Universal Robots PolyScope program: despellatizing.urp

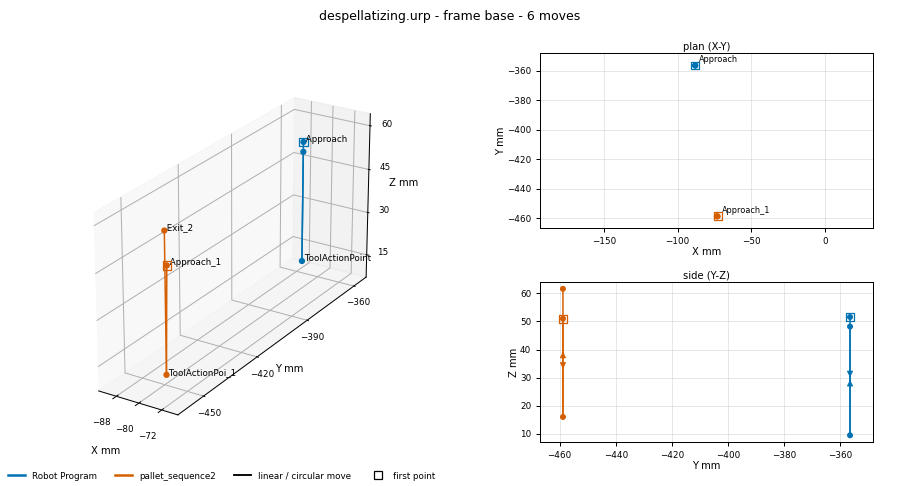
[picture p0: tool path of despellatizing.urp in frame base, 6 of 6 moves have a stored position in this frame; points joined in program order, loops and branches not executed]
Program despellatizing (installation=default ventosa directory=/programs/usbdisk/Ventosa-paleta createdIn=5.12.1.1101497 lastSavedIn=5.12.1.1101497 robotSerialNumber=20225300640)
Calibrated DH parameters: a=[-0.000125, -0.240482, -0.204397, 0.000169, -0.000135, 0]; d=[0.152056, 4.760815, 12.138494, -16.768367, 0.085457, 0.092357]; alpha=[1.570863, 0.008548, 0.003635, 1.571424, -1.571918, 0]; deltaTheta=[0, 0.167622, 0.124346, -0.291972, 0.000034, 0]
BeforeStart
  SafeHome (positionOptionType=SPEED_AND_ACCELERATION speed=1.047198 acceleration=1.396263 nextMotionTime=2)
  cnt_obj := 0
Robot Program (runOnlyOnce=true)
  Loop While (checkContinuously=false) expression=cnt_obj<2
    URCap Palletizing (polyscope-pallet-impl, Universal Robots) dataModel(palletFeature=Base, isPalletizing=false, Variable(key=name, variable(name=Pallet_1)), Variable(key=globalCountingVariable, variable(name=Pallet_1_cnt, initializeExpression=1)), Variable(key=layerNumberVariable, variable(name=Pallet_1_lno, initializeExpression=1)), Variable(key=layerCountingVariable, variable(name=Pallet_1_lct, initializeExpression=1)), Variable(key=handleSeparatorVariable, variable(name=Pallet_1_sep, initializeExpression=False)), Variable(key=totalCountVariable, variable(name=Pallet_1_tct, initializeExpression=1)), Variable(key=referencePoint, variable(featureName=referencePoint)), Variable(key=separatorPoint, variable(featureName=separatorPoint)), Length(key=objectHeight value=0.02 unit=M)); state(isChildrenLocked=true)
      URCap Patterns (polyscope-pallet-impl, Universal Robots) state(isChildrenLocked=true)
        URCap Pattern (polyscope-pallet-impl, Universal Robots) dataModel(UUID=4f81d8ba-079c-47d5-9963-bf25775c8eb8, patternType=LINE, objects=3, Variable(key=nameVariable, variable(name=Line_Pattern_1))); state(isChildrenLocked=true)
          URCap Item (polyscope-pallet-impl, Universal Robots) dataModel(UUID=1e3ca6f4-2eef-47f5-9254-e2ca323da8c7, patternType=LINE, index=0, calibrationDeltaTheta=[-4.022425301349053E-7, 0.1676224840059082, 0.12434612800300923, -0.29197201232783093, 3.427063592260221E-5, -2.1055269264214083E-9], calibrationA=[-1.2536318386722594E-4, -0.24048217598078755, -0.20439712606180582, 1.6856812341359539E-4, -1.3512489031768148E-4, 0.0], calibrationD=[0.1520559623222255, 4.760815016703785, 12.138493934059257, -16.768366633975226, 0.08545691164632878, 0.09235657960129308], calibrationAlpha=[1.570862629498801, 0.008547662301921876, 0.0036353825850200293, 1.5714242532258311, -1.5719182813352055, 0.0], calibrationJointChecksum=[-1442419114, -1443167645, -1459096000, -1465254611, -1461595521, -1465327861], calibrationStatus=2, calibrationValidChecksum=true, baseToFeature=[0.0, 0.0, 0.0, 0.0, 0.0, 0.0], TCPOffset=[-3.1361648691191624E-6, -7.165658321095503E-6, 0.14500622770334937, -3.159826595633942E-6, 1.3472828827308191E-6, -1.5977345697242604E-5], Variable(key=variable, variable(name=StartItem_1)), JointPositions(key=jointpositions, JointPosition(key=[1], Angle(key=pos value=0.956268 unit=RAD)), JointPosition(key=[2], Angle(key=pos value=-1.20615 unit=RAD)), JointPosition(key=[3], Angle(key=pos value=1.878719 unit=RAD)), JointPosition(key=[4], Angle(key=pos value=-2.25283 unit=RAD)), JointPosition(key=[5], Angle(key=pos value=-1.545112 unit=RAD)), JointPosition(key=[6], Angle(key=pos value=-0.610524 unit=RAD))))
          URCap Item (polyscope-pallet-impl, Universal Robots) dataModel(UUID=6f3f843f-6f96-4607-877d-a96ceec1e152, patternType=LINE, index=1, calibrationDeltaTheta=[-4.022425301349053E-7, 0.1676224840059082, 0.12434612800300923, -0.29197201232783093, 3.427063592260221E-5, -2.1055269264214083E-9], calibrationA=[-1.2536318386722594E-4, -0.24048217598078755, -0.20439712606180582, 1.6856812341359539E-4, -1.3512489031768148E-4, 0.0], calibrationD=[0.1520559623222255, 4.760815016703785, 12.138493934059257, -16.768366633975226, 0.08545691164632878, 0.09235657960129308], calibrationAlpha=[1.570862629498801, 0.008547662301921876, 0.0036353825850200293, 1.5714242532258311, -1.5719182813352055, 0.0], calibrationJointChecksum=[-1442419114, -1443167645, -1459096000, -1465254611, -1461595521, -1465327861], calibrationStatus=2, calibrationValidChecksum=true, baseToFeature=[0.0, 0.0, 0.0, 0.0, 0.0, 0.0], TCPOffset=[-8.933406672184674E-6, 6.908638976621528E-6, 0.14500541786871218, -1.4995112137550501E-5, -1.239510916399233E-6, -2.697305733370411E-5], Variable(key=variable, variable(name=EndItem_1)), JointPositions(key=jointpositions, JointPosition(key=[1], Angle(key=pos value=1.450295 unit=RAD)), JointPosition(key=[2], Angle(key=pos value=-1.189136 unit=RAD)), JointPosition(key=[3], Angle(key=pos value=1.845346 unit=RAD)), JointPosition(key=[4], Angle(key=pos value=-2.243967 unit=RAD)), JointPosition(key=[5], Angle(key=pos value=-1.548882 unit=RAD)), JointPosition(key=[6], Angle(key=pos value=-0.116345 unit=RAD))))
      URCap Layers (polyscope-pallet-impl, Universal Robots) dataModel(separators=[false], selectedPatterns=[4f81d8ba-079c-47d5-9963-bf25775c8eb8])
      URCap At Each Item (polyscope-pallet-impl, Universal Robots) dataModel(selectedPattern=4f81d8ba-079c-47d5-9963-bf25775c8eb8, selectedPosition=1e3ca6f4-2eef-47f5-9254-e2ca323da8c7, Approach_calibrationDeltaTheta=[-4.022425301349053E-7, 0.1676224840059082, 0.12434612800300923, -0.29197201232783093, 3.427063592260221E-5, -2.1055269264214083E-9], Approach_calibrationA=[-1.2536318386722594E-4, -0.24048217598078755, -0.20439712606180582, 1.6856812341359539E-4, -1.3512489031768148E-4, 0.0], Approach_calibrationD=[0.1520559623222255, 4.760815016703785, 12.138493934059257, -16.768366633975226, 0.08545691164632878, 0.09235657960129308], Approach_calibrationAlpha=[1.570862629498801, 0.008547662301921876, 0.0036353825850200293, 1.5714242532258311, -1.5719182813352055, 0.0], Approach_calibrationJointChecksum=[-1442419114, -1443167645, -1459096000, -1465254611, -1461595521, -1465327861], Approach_calibrationStatus=2, Approach_calibrationValidChecksum=true, Approach_baseToFeature=[0.0, 0.0, 0.0, 0.0, 0.0, 0.0], Approach_TCPOffset=[-9.367263874154874E-6, -3.571446355488117E-6, 0.1449987796699207, 2.480276054203756E-5, -1.6285190499819042E-5, -2.849487153099717E-6], Exit_calibrationDeltaTheta=[-4.022425301349053E-7, 0.1676224840059082, 0.12434612800300923, -0.29197201232783093, 3.427063592260221E-5, -2.1055269264214083E-9], Exit_calibrationA=[-1.2536318386722594E-4, -0.24048217598078755, -0.20439712606180582, 1.6856812341359539E-4, -1.3512489031768148E-4, 0.0], Exit_calibrationD=[0.1520559623222255, 4.760815016703785, 12.138493934059257, -16.768366633975226, 0.08545691164632878, 0.09235657960129308], Exit_calibrationAlpha=[1.570862629498801, 0.008547662301921876, 0.0036353825850200293, 1.5714242532258311, -1.5719182813352055, 0.0], Exit_calibrationJointChecksum=[-1442419114, -1443167645, -1459096000, -1465254611, -1461595521, -1465327861], Exit_calibrationStatus=2, Exit_calibrationValidChecksum=true, Exit_baseToFeature=[0.0, 0.0, 0.0, 0.0, 0.0, 0.0], Exit_TCPOffset=[-1.637346477856294E-5, 4.478754114078942E-6, 0.14501055095189264, -4.558640450482124E-5, -2.3885119760789442E-6, -5.824444254552941E-5], currentWizardState=LANDING, Pose(key=refBaseToFeature, Position(key=posePosition, Length(key=X value=0 unit=M), Length(key=Y value=0 unit=M), Length(key=Z value=0 unit=M)), Rotation(key=poseRotation, Angle(key=RX value=0 unit=RAD), Angle(key=RY value=0 unit=RAD), Angle(key=RZ value=0 unit=RAD))), Pose(key=refPose, Position(key=posePosition, Length(key=X value=-0.087998 unit=M), Length(key=Y value=-0.356588 unit=M), Length(key=Z value=0.009445 unit=M)), Rotation(key=poseRotation, Angle(key=RX value=0.013823 unit=RAD), Angle(key=RY value=3.130534 unit=RAD), Angle(key=RZ value=-0.028056 unit=RAD))), JointPositions(key=Approach_jointpositions, JointPosition(key=[1], Angle(key=pos value=0.956543 unit=RAD)), JointPosition(key=[2], Angle(key=pos value=-1.303654 unit=RAD)), JointPosition(key=[3], Angle(key=pos value=1.781977 unit=RAD)), JointPosition(key=[4], Angle(key=pos value=-2.05857 unit=RAD)), JointPosition(key=[5], Angle(key=pos value=-1.54531 unit=RAD)), JointPosition(key=[6], Angle(key=pos value=-0.611111 unit=RAD))), JointPositions(key=Exit_jointpositions, JointPosition(key=[1], Angle(key=pos value=0.956524 unit=RAD)), JointPosition(key=[2], Angle(key=pos value=-1.296966 unit=RAD)), JointPosition(key=[3], Angle(key=pos value=1.79099 unit=RAD)), JointPosition(key=[4], Angle(key=pos value=-2.074272 unit=RAD)), JointPosition(key=[5], Angle(key=pos value=-1.545298 unit=RAD)), JointPosition(key=[6], Angle(key=pos value=-0.611064 unit=RAD))))
        URCap Generated Movements (polyscope-pallet-impl, Universal Robots) state(isChildrenLocked=true)
          MoveJ speed 60 deg/s, acceleration 80 deg/s^2 (useActiveTCP=true) feature=referencePoint
            Waypoint Approach: TCP in base x=-87.988 y=-356.591 z=51.588 mm, rx=0.0138 ry=3.1305 rz=-0.0281 rad; joints [55.219, -48.655, 112.12, -154.019, -88.483, -34.404] deg; TCP offset x=0 y=0 z=0 mm, rx=0 ry=0 rz=0 rad; feature pose in base x=-87.998 y=-356.588 z=9.445 mm, rx=0.0138 ry=3.1305 rz=-0.0281 rad
          MoveL speed 250 mm/s, acceleration 1200 mm/s^2 (useActiveTCP=true) feature(featureName=referencePoint)
            Waypoint ToolActionPoint: TCP in base x=-87.998 y=-356.588 z=9.445 mm, rx=0.0138 ry=3.1305 rz=-0.0281 rad; joints [55.202, -38.806, 110.643, -162.392, -88.468, -34.349] deg; TCP offset x=0 y=0 z=0 mm, rx=0 ry=0 rz=0 rad
          Folder Tool action
            URCap Vacuum (Robotiq_Grippers, Robotiq Inc.) dataModel(Vacuum.Command.PumpAutoCloseDelayInMilliseconds=3000, Vacuum.Command.ShutOffDistance=5.0)
          MoveL speed 250 mm/s, acceleration 1200 mm/s^2 (useActiveTCP=true) feature(featureName=referencePoint)
            Waypoint Exit_1: TCP in base x=-87.981 y=-356.583 z=48.176 mm, rx=0.0137 ry=3.1305 rz=-0.028 rad; joints [55.219, -47.88, 112.079, -154.751, -88.485, -34.402] deg; TCP offset x=0 y=0 z=0 mm, rx=0 ry=0 rz=0 rad
            URCap Grip Check (Robotiq_Grippers, Robotiq Inc.) dataModel(ObjectDetectedKey=true, DimensionValidationKey=false, DimensionKey=100.0, DimensionDimensionPositiveGapKey=5.0, DimensionNegativeGapKey=5.0, GripperIdKey=1, ModelDefinedKey=true); state(isChildrenLocked=true)
              URCap If (Robotiq_Grippers, Robotiq Inc.)
                Call pallet_sequence2
                cnt_obj := cnt_obj+1
              URCap Else (Robotiq_Grippers, Robotiq Inc.)
                URCap Vacuum (Robotiq_Grippers, Robotiq Inc.) dataModel(Vacuum.Command.PumpAutoCloseDelayInMilliseconds=3000, Vacuum.Command.ShutOffDistance=5.0, Vacuum.Command.Action=1)
  SafeHome (positionOptionType=SPEED_AND_ACCELERATION speed=1.047198 acceleration=1.396263 nextMotionTime=2)
SubProgram -> pallet_sequence2
SubProgram pallet_sequence2 (keepSynchronizedWithDisk=false)
  URCap Palletizing (polyscope-pallet-impl, Universal Robots) dataModel(palletFeature=Base, isPalletizing=true, Variable(key=name, variable(name=Pallet_2)), Variable(key=globalCountingVariable, variable(name=Pallet_2_cnt, initializeExpression=1)), Variable(key=layerNumberVariable, variable(name=Pallet_2_lno, initializeExpression=1)), Variable(key=layerCountingVariable, variable(name=Pallet_2_lct, initializeExpression=1)), Variable(key=handleSeparatorVariable, variable(name=Pallet_2_sep, initializeExpression=False)), Variable(key=totalCountVariable, variable(name=Pallet_2_tct, initializeExpression=1)), Variable(key=referencePoint, variable(featureName=referencePoin_1)), Variable(key=separatorPoint, variable(featureName=separatorPoin_1)), Length(key=objectHeight value=0.02 unit=M)); state(isChildrenLocked=true)
    URCap Patterns (polyscope-pallet-impl, Universal Robots) state(isChildrenLocked=true)
      URCap Pattern (polyscope-pallet-impl, Universal Robots) dataModel(UUID=6eecd687-f34c-4585-a3fc-93ce3e107647, patternType=LINE, objects=2, Variable(key=nameVariable, variable(name=Line_Pattern_2))); state(isChildrenLocked=true)
        URCap Item (polyscope-pallet-impl, Universal Robots) dataModel(UUID=5ae76496-7a2a-494b-879e-71bc1cc3e574, patternType=LINE, index=0, calibrationDeltaTheta=[-4.022425301349053E-7, 0.1676224840059082, 0.12434612800300923, -0.29197201232783093, 3.427063592260221E-5, -2.1055269264214083E-9], calibrationA=[-1.2536318386722594E-4, -0.24048217598078755, -0.20439712606180582, 1.6856812341359539E-4, -1.3512489031768148E-4, 0.0], calibrationD=[0.1520559623222255, 4.760815016703785, 12.138493934059257, -16.768366633975226, 0.08545691164632878, 0.09235657960129308], calibrationAlpha=[1.570862629498801, 0.008547662301921876, 0.0036353825850200293, 1.5714242532258311, -1.5719182813352055, 0.0], calibrationJointChecksum=[-1442419114, -1443167645, -1459096000, -1465254611, -1461595521, -1465327861], calibrationStatus=2, calibrationValidChecksum=true, baseToFeature=[0.0, 0.0, 0.0, 0.0, 0.0, 0.0], TCPOffset=[-3.825552644387553E-6, 2.2159503549903925E-5, 0.14498391099687513, -9.769649068358888E-7, 3.7748736814289966E-6, 9.716702353280994E-5], Variable(key=variable, variable(name=StartItem_2)), JointPositions(key=jointpositions, JointPosition(key=[1], Angle(key=pos value=1.140796 unit=RAD)), JointPosition(key=[2], Angle(key=pos value=-0.843807 unit=RAD)), JointPosition(key=[3], Angle(key=pos value=1.21922 unit=RAD)), JointPosition(key=[4], Angle(key=pos value=-1.930381 unit=RAD)), JointPosition(key=[5], Angle(key=pos value=-1.548959 unit=RAD)), JointPosition(key=[6], Angle(key=pos value=-1.966878 unit=RAD))))
        URCap Item (polyscope-pallet-impl, Universal Robots) dataModel(UUID=8c4953bf-a7e4-4ce7-9c88-c1d62482faca, patternType=LINE, index=1, calibrationDeltaTheta=[-4.022425301349053E-7, 0.1676224840059082, 0.12434612800300923, -0.29197201232783093, 3.427063592260221E-5, -2.1055269264214083E-9], calibrationA=[-1.2536318386722594E-4, -0.24048217598078755, -0.20439712606180582, 1.6856812341359539E-4, -1.3512489031768148E-4, 0.0], calibrationD=[0.1520559623222255, 4.760815016703785, 12.138493934059257, -16.768366633975226, 0.08545691164632878, 0.09235657960129308], calibrationAlpha=[1.570862629498801, 0.008547662301921876, 0.0036353825850200293, 1.5714242532258311, -1.5719182813352055, 0.0], calibrationJointChecksum=[-1442419114, -1443167645, -1459096000, -1465254611, -1461595521, -1465327861], calibrationStatus=2, calibrationValidChecksum=true, baseToFeature=[0.0, 0.0, 0.0, 0.0, 0.0, 0.0], TCPOffset=[7.1373890455639355E-6, 1.5658113228025905E-5, 0.14500116724169027, 4.767946296077085E-6, -4.537083107082065E-6, -6.555073351997114E-6], Variable(key=variable, variable(name=EndItem_2)), JointPositions(key=jointpositions, JointPosition(key=[1], Angle(key=pos value=1.441147 unit=RAD)), JointPosition(key=[2], Angle(key=pos value=-0.848924 unit=RAD)), JointPosition(key=[3], Angle(key=pos value=1.234156 unit=RAD)), JointPosition(key=[4], Angle(key=pos value=-1.944504 unit=RAD)), JointPosition(key=[5], Angle(key=pos value=-1.544494 unit=RAD)), JointPosition(key=[6], Angle(key=pos value=-1.666434 unit=RAD))))
    URCap Layers (polyscope-pallet-impl, Universal Robots) dataModel(separators=[false], selectedPatterns=[6eecd687-f34c-4585-a3fc-93ce3e107647])
    URCap At Each Item (polyscope-pallet-impl, Universal Robots) dataModel(selectedPattern=6eecd687-f34c-4585-a3fc-93ce3e107647, selectedPosition=5ae76496-7a2a-494b-879e-71bc1cc3e574, Approach_calibrationDeltaTheta=[-4.022425301349053E-7, 0.1676224840059082, 0.12434612800300923, -0.29197201232783093, 3.427063592260221E-5, -2.1055269264214083E-9], Approach_calibrationA=[-1.2536318386722594E-4, -0.24048217598078755, -0.20439712606180582, 1.6856812341359539E-4, -1.3512489031768148E-4, 0.0], Approach_calibrationD=[0.1520559623222255, 4.760815016703785, 12.138493934059257, -16.768366633975226, 0.08545691164632878, 0.09235657960129308], Approach_calibrationAlpha=[1.570862629498801, 0.008547662301921876, 0.0036353825850200293, 1.5714242532258311, -1.5719182813352055, 0.0], Approach_calibrationJointChecksum=[-1442419114, -1443167645, -1459096000, -1465254611, -1461595521, -1465327861], Approach_calibrationStatus=2, Approach_calibrationValidChecksum=true, Approach_baseToFeature=[0.0, 0.0, 0.0, 0.0, 0.0, 0.0], Approach_TCPOffset=[7.60713690806103E-6, -2.2154056772069608E-5, 0.14499029150698028, 2.9459734422612152E-5, 3.3660089335491905E-5, -1.1450730779261408E-5], Exit_calibrationDeltaTheta=[-4.022425301349053E-7, 0.1676224840059082, 0.12434612800300923, -0.29197201232783093, 3.427063592260221E-5, -2.1055269264214083E-9], Exit_calibrationA=[-1.2536318386722594E-4, -0.24048217598078755, -0.20439712606180582, 1.6856812341359539E-4, -1.3512489031768148E-4, 0.0], Exit_calibrationD=[0.1520559623222255, 4.760815016703785, 12.138493934059257, -16.768366633975226, 0.08545691164632878, 0.09235657960129308], Exit_calibrationAlpha=[1.570862629498801, 0.008547662301921876, 0.0036353825850200293, 1.5714242532258311, -1.5719182813352055, 0.0], Exit_calibrationJointChecksum=[-1442419114, -1443167645, -1459096000, -1465254611, -1461595521, -1465327861], Exit_calibrationStatus=2, Exit_calibrationValidChecksum=true, Exit_baseToFeature=[0.0, 0.0, 0.0, 0.0, 0.0, 0.0], Exit_TCPOffset=[1.6192892542399306E-6, -3.7896869635595243E-6, 0.14499457199851368, -4.248067248152122E-6, 8.005632300632978E-6, -3.5079730383509784E-5], currentWizardState=LANDING, Pose(key=refBaseToFeature, Position(key=posePosition, Length(key=X value=0 unit=M), Length(key=Y value=0 unit=M), Length(key=Z value=0 unit=M)), Rotation(key=poseRotation, Angle(key=RX value=0 unit=RAD), Angle(key=RY value=0 unit=RAD), Angle(key=RZ value=0 unit=RAD))), Pose(key=refPose, Position(key=posePosition, Length(key=X value=-0.073385 unit=M), Length(key=Y value=-0.45883 unit=M), Length(key=Z value=0.015967 unit=M)), Rotation(key=poseRotation, Angle(key=RX value=-2.164921 unit=RAD), Angle(key=RY value=2.248539 unit=RAD), Angle(key=RZ value=-0.008283 unit=RAD))), JointPositions(key=Approach_jointpositions, JointPosition(key=[1], Angle(key=pos value=1.124632 unit=RAD)), JointPosition(key=[2], Angle(key=pos value=-0.879331 unit=RAD)), JointPosition(key=[3], Angle(key=pos value=1.110265 unit=RAD)), JointPosition(key=[4], Angle(key=pos value=-1.785693 unit=RAD)), JointPosition(key=[5], Angle(key=pos value=-1.549145 unit=RAD)), JointPosition(key=[6], Angle(key=pos value=-1.983713 unit=RAD))), JointPositions(key=Exit_jointpositions, JointPosition(key=[1], Angle(key=pos value=1.12331 unit=RAD)), JointPosition(key=[2], Angle(key=pos value=-0.889114 unit=RAD)), JointPosition(key=[3], Angle(key=pos value=1.076368 unit=RAD)), JointPosition(key=[4], Angle(key=pos value=-1.741995 unit=RAD)), JointPosition(key=[5], Angle(key=pos value=-1.54915 unit=RAD)), JointPosition(key=[6], Angle(key=pos value=-1.985238 unit=RAD))))
      URCap Generated Movements (polyscope-pallet-impl, Universal Robots) state(isChildrenLocked=true)
        MoveJ speed 60 deg/s, acceleration 80 deg/s^2 (useActiveTCP=true) feature=referencePoin_1
          Waypoint Approach_1: TCP in base x=-72.722 y=-458.827 z=50.992 mm, rx=-2.1649 ry=2.2485 rz=-0.0084 rad; joints [64.652, -33.913, 75.624, -130.799, -88.746, -113.252] deg; TCP offset x=0 y=0 z=0 mm, rx=0 ry=0 rz=0 rad; feature pose in base x=-73.385 y=-458.83 z=15.967 mm, rx=-2.1649 ry=2.2485 rz=-0.0083 rad
        MoveL speed 250 mm/s, acceleration 1200 mm/s^2 (useActiveTCP=true) feature(featureName=referencePoin_1)
          Waypoint ToolActionPoi_1: TCP in base x=-73.385 y=-458.83 z=15.967 mm, rx=-2.1649 ry=2.2485 rz=-0.0083 rad; joints [64.564, -27.94, 74.6, -135.747, -88.746, -113.283] deg; TCP offset x=0 y=0 z=0 mm, rx=0 ry=0 rz=0 rad
        Folder Tool action
          URCap Vacuum (Robotiq_Grippers, Robotiq Inc.) dataModel(Vacuum.Command.Action=1, Vacuum.Command.PumpAutoCloseDelayInMilliseconds=3000, Vacuum.Command.ShutOffDistance=5.0)
        MoveL speed 250 mm/s, acceleration 1200 mm/s^2 (useActiveTCP=true) feature(featureName=referencePoin_1)
          Waypoint Exit_2: TCP in base x=-73.381 y=-458.831 z=61.614 mm, rx=-2.165 ry=2.2485 rz=-0.0083 rad; joints [64.58, -35.583, 75.596, -129.1, -88.751, -113.342] deg; TCP offset x=0 y=0 z=0 mm, rx=0 ry=0 rz=0 rad
